DATA_BLOCK "Zne09_DB"
{ S7_Optimized_Access := 'TRUE' }
VERSION : 0.1
NON_RETAIN
"Zne09"

BEGIN

END_DATA_BLOCK

